{attribute 'TcGenerated'}
{attribute 'no-analysis'}
{attribute 'linkalways'}
// This function has been automatically generated from the project information.
VAR_GLOBAL CONSTANT
	{attribute 'const_non_replaced'}
	stLibVersion_Tc_Utilities : ST_LibVersion := (iMajor := 0, iMinor := 0, iBuild := 0, iRevision := 1, nFlags := 0, sVersion := '0.0.0.1');
END_VAR

(* stored: Version 1.1.0.1, ProductVersion 3.1.4024.12
   GVL Global_Version: Id {d6611707-3d65-4502-99b8-e173a1416047} *)
